PROGRAM notes
VAR
END_VAR

(*
To add a shortcut:
1. Tools -> Options -> Environment -> Keyboard
2. Search for functions
	Example: Logintonone
3. Press shortcut keys -> Assign



Change variables while running program
1. Add value to 'prepared values' column
2. 'Write values' (top right)
	Shortcut -> Alt-W 
	
	
Shortcuts:
Write values: Alt-W
Login: Alt-X
Logout: Alt-Z
Input assistant: F2 (or right click in program section

Terms:
Rising edge: when input goes from low to high
Falling edge: opposite of above

Notes:
Libraries are in PLC -> references
Set reserved/shared cores in SYSTEM-> Real-Time
Set run speed (cycles) in PLC -> PlcTask, or SYSTEM -> Tasks -> PlcTask
Multi line comments  -> (**)
Regular comment -> /

if statement:
IF {condition} THEN
	{body}
END_IF

loop:
FOR variable := start-value TO end-value [ BY step-value ] DO
    statement;
    statement;
    ..
    statement;
END_FOR;

function:
Function CalcStdDev : LREAL
var_input v1,v2,v3,v4 : LREAL; end_var

var 
    SumOfSquares : LREAL;
    Mean : LREAL;
end_var

    (* Calculate the mean *)
    Mean := (v1 + v2 + v3 + v4) / 4;

    (* Calculate the standard deviation *)
    SumOfSquares := (v1 - Mean) ** 2 +
                (v2 - Mean) ** 2 +
                (v3 - Mean) ** 2 +
                (v4 - Mean) ** 2;

    CalcStdDev := sqrt( SumOfSquares / 4 );
End_Function

*)

END_PROGRAM

(* stored: Version 1.1.0.1, ProductVersion 3.1.4024.13
   POU notes: Id {435b32a7-83f5-464f-b5b0-8632d772ace8}, SpecialFunc None *)
